FUNCTION_BLOCK FB_Timestamp
VAR_INPUT
END_VAR
VAR_OUTPUT
END_VAR
VAR
	nTimestamp:			ULINT;
END_VAR

METHOD PUBLIC M_Create
VAR_INPUT
END_VAR
nTimestamp:= F_GetSystemTime();
END_METHOD

METHOD PUBLIC M_ToSTRING : String(255)
VAR_INPUT
END_VAR
SYSTEMTIME_TO_STRING(M_ToTIMESTRUCT());
END_METHOD

METHOD PUBLIC M_ToTIMESTRUCT : TIMESTRUCT
VAR_INPUT
END_VAR
M_ToTIMESTRUCT:= FILETIME_TO_SYSTEMTIME(nTimestamp);
END_METHOD

END_FUNCTION_BLOCK

(* stored: Version 1.1.0.1, ProductVersion 3.1.4024.12
   POU FB_Timestamp: Id {83d29445-3227-061e-34fb-c2c7ad5219b7}, SpecialFunc None
   Method M_Create: Id {ccdea776-6ef9-0715-3563-9fac1e94846f}
   Method M_ToSTRING: Id {62a96ac9-3bcc-07ab-36d0-e2a2f9371537}
   Method M_ToTIMESTRUCT: Id {21021426-75a6-03ef-1f46-d69b579da397} *)
